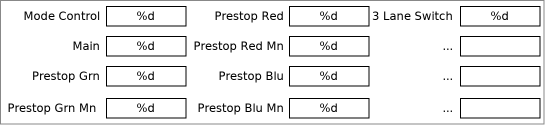
VISUALIZATION StateDisplay  // 545x125
    Rectangle (187,66 100x20), "Prestop Blu"
    Rectangle (289,66 80x20), "%d", text variable: Stn051_14_ReturnLnSwPrestopBlu.fbConvStop.Local.State
    Rectangle (356,66 100x20), "..."
    Rectangle (460,66 80x20)
    Rectangle (3,66 100x20), "Prestop Grn"
    Rectangle (106,66 80x20), "%d", text variable: Stn051_10_ReturnLnSwPrestopGrn.fbConvStop.Local.State
    Rectangle (3,6 100x20), "Mode Control"
    Rectangle (106,6 80x20), "%d", text variable: Stn051_00_ModeControl.Local.State
    Rectangle (187,6 100x20), "Prestop Red"
    Rectangle (289,6 80x20), "%d", text variable: Stn051_12_ReturnLnSwPrestopRed.fbConvStop.Local.State
    Rectangle (356,6 100x20), "3 Lane Switch"
    Rectangle (460,6 80x20), "%d", text variable: Stn051_16_ReturnLnSw.fb3LaneSwitchMain.Local.State
    Rectangle (23,36 80x20), "Main"
    Rectangle (106,36 80x20), "%d", text variable: Stn051_05_StnMain.Local.State
    Rectangle (356,36 100x20), "..."
    Rectangle (460,36 80x20)
    Rectangle (187,36 100x20), "Prestop Red Mn"
    Rectangle (289,36 80x20), "%d", text variable: Stn051_13_ReturnLnSwPrestopMainRed.fbWorkStopMainLnSw.Local.State
    Rectangle (187,98 100x20), "Prestop Blu Mn"
    Rectangle (289,98 80x20), "%d", text variable: Stn051_15_ReturnLnSwPrestopMainBlu.fbWorkStopMainLnSw.Local.State
    Rectangle (4,98 99x20), "Prestop Grn Mn"
    Rectangle (106,98 80x20), "%d", text variable: Stn051_11_ReturnLnSwPrestopMainGrn.fbWorkStopMainLnSw.Local.State
    Rectangle (370,98 86x20), "..."
    Rectangle (460,98 80x20)
END_VISUALIZATION

(* stored: Version 1.1.0.1, ProductVersion 3.1.4024.6
   Visu StateDisplay: Id {9f29c517-ab78-4783-9711-5d4f9690602e} *)
